FUNCTION_BLOCK FB_Linked_List_Stack IMPLEMENTS I_Stack
VAR_INPUT
END_VAR
VAR_OUTPUT
END_VAR
VAR
END_VAR

{warning 'add method implementation '}
METHOD Peek : T_DATA_TYPE
END_METHOD

{warning 'add method implementation '}
METHOD Pop
END_METHOD

{warning 'add method implementation '}
METHOD Push
VAR_INPUT
	Data	: T_DATA_TYPE;
END_VAR
END_METHOD

{warning 'add method implementation '}
METHOD Show
END_METHOD

END_FUNCTION_BLOCK

(* stored: Version 1.1.0.1, ProductVersion 3.1.4024.4
   POU FB_Linked_List_Stack: Id {2c59cdc2-33c5-4868-bca4-01c093a816a0}, SpecialFunc None
   Method Peek: Id {c2639508-4e31-4b41-ba23-49c69940227c}
   Method Pop: Id {859ccdaa-4bef-4e52-91c9-55ee71ff56a8}
   Method Push: Id {bedbe239-212f-42b1-8e7c-4d2a523feac0}
   Method Show: Id {24bc1739-b5a7-45aa-816d-caa104c39755} *)
